// TIA Portal V17 export
// export: Created 2024-09-02T12:49:58.6540068Z, ExportSetting WithDefaults, DisplayName Totally Integrated Automation Portal, DisplayVersion V17, DisplayName TIA Portal Openness, DisplayVersion V17, DisplayName TIA Portal Version Control Interface, DisplayVersion V17, DisplayName STEP 7 Professional, DisplayVersion V17, DisplayName STEP 7 Safety, DisplayVersion V17, DisplayName WinCC Professional, DisplayVersion V17
ORGANIZATION_BLOCK "OB_Cycle_Extension"   // OB1, LAD, ProgramCycle
TITLE = Cyclic program processing of the VW additional blocks / "Main Program Sweep (Cycle)" / Zyklische Programmbearbeitung der VW Zusatzbausteine
{ S7_Optimized_Access := 'TRUE' }
VERSION : 0.1
// stored: AutoNumber true, IsIECCheckEnabled false, SetENOAutomatically false
   VAR_INPUT
      Initial_Call : Bool;   // Initial call of this OB
      Remanence : Bool;   // =True, if remanent data are available
   END_VAR
   VAR_TEMP
      RET_VAL_WR_LOC_T : Int;
   END_VAR
BEGIN

REGION Network 1: Call FB Machine load and shift model / Aufruf FB Machinenauslastung und Schichtmodell
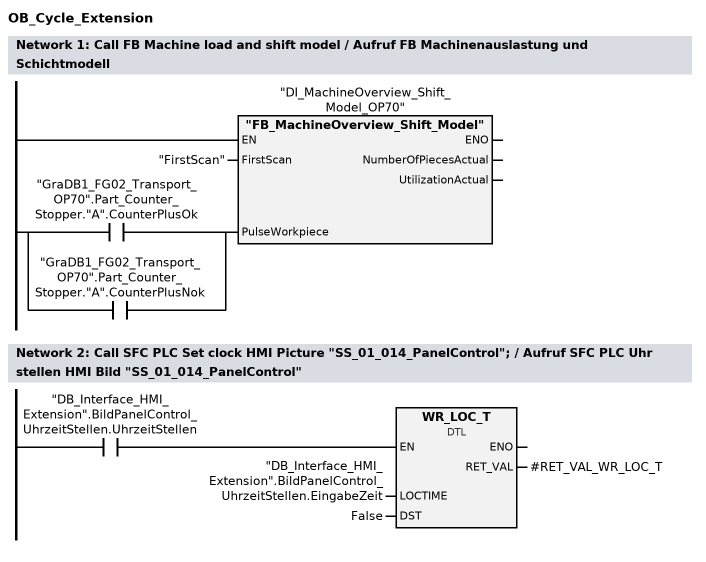
   RUNG wire#powerrail
      "DI_MachineOverview_Shift_Model_OP70"(PulseWorkpiece := wire#w1, FirstScan := "FirstScan", NumberOfPiecesActual =>, UtilizationActual =>)
   END_RUNG
   RUNG wire#powerrail
      Contact( "GraDB1_FG02_Transport_OP70".Part_Counter_Stopper."A".CounterPlusOk )
   END_RUNG wire#w1
   RUNG wire#powerrail
      Contact( "GraDB1_FG02_Transport_OP70".Part_Counter_Stopper."A".CounterPlusNok )
   END_RUNG wire#w1
   // the same network as SCL:
   "DI_MachineOverview_Shift_Model_OP70"(FirstScan := "FirstScan",   // "FB_MachineOverview_Shift_Model"
                           PulseWorkpiece := "GraDB1_FG02_Transport_OP70".Part_Counter_Stopper."A".CounterPlusOk OR "GraDB1_FG02_Transport_OP70".Part_Counter_Stopper."A".CounterPlusNok);
END_REGION

REGION Network 2: Call SFC PLC Set clock HMI Picture "SS_01_014_PanelControl"; / Aufruf SFC PLC Uhr stellen HMI Bild "SS_01_014_PanelControl"
   RUNG wire#powerrail
      Contact( "DB_Interface_HMI_Extension".BildPanelControl_UhrzeitStellen.UhrzeitStellen )
      { S7_Templates := "loctime_type := DTL" } WR_LOC_T(LOCTIME := "DB_Interface_HMI_Extension".BildPanelControl_UhrzeitStellen.EingabeZeit, DST := False, Ret_Val => #RET_VAL_WR_LOC_T)
   END_RUNG
   // the same network as SCL:
   IF "DB_Interface_HMI_Extension".BildPanelControl_UhrzeitStellen.UhrzeitStellen THEN
       #RET_VAL_WR_LOC_T := WR_LOC_T(LOCTIME := "DB_Interface_HMI_Extension".BildPanelControl_UhrzeitStellen.EingabeZeit,
                               DST := False);
   END_IF;
END_REGION
END_ORGANIZATION_BLOCK
